TYPE U_Estop :
UNION
	Pos	:E_EStop;	
	IO 	:ST_EstopIO;
END_UNION
END_TYPE

(* stored: Version 1.1.0.1
   DUT U_Estop: Id {891a96e7-55b8-4bcf-8053-9416c82b7dc9} *)
